FUNCTION_BLOCK RequestOrchestrationOpcUa (* Request Orchestration Function Block using OPC UA *)
  (* Standard: 61499-2; Description: Copyright (c) 2019 fortiss GmbH This program and the accompanying materials are made available under the terms of the Eclipse Public License 2.0 which is available at https://www.eclipse.org/legal/epl-2.0/ SPDX-License-Identifier: EPL-2.0 *)
  (* Version 1.0, 2019-09-17, Jose Cabral, fortiss GmbH *)
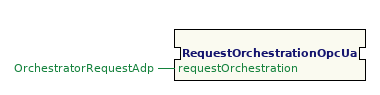
  SOCKETS
    requestOrchestration : OrchestratorRequestAdp; (* Request orchestration adapter *)
  END_SOCKETS
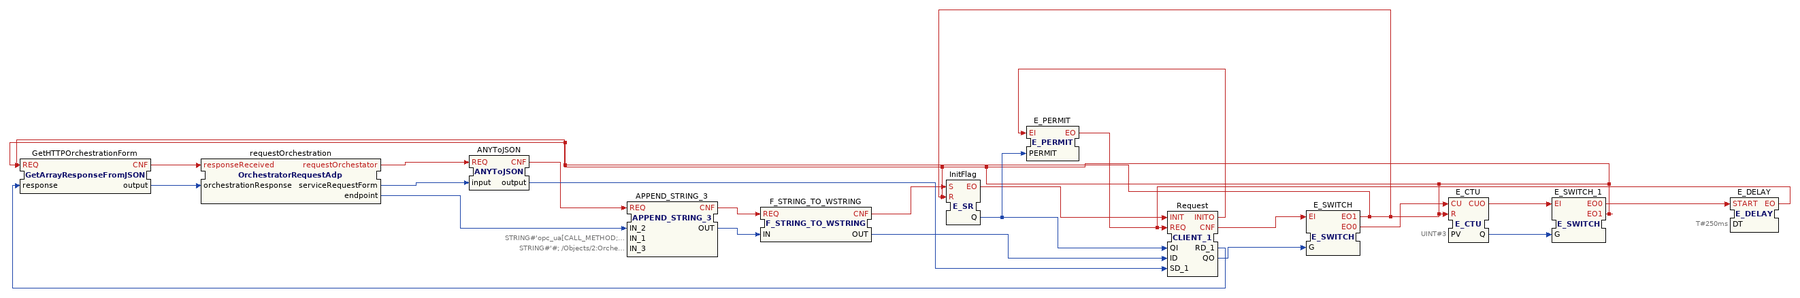
  FBS
    APPEND_STRING_3 : APPEND_STRING_3(IN_1 := STRING#'opc_ua[CALL_METHOD; ', IN_3 := STRING#'#; /Objects/2:Orchestrator/2:orchestration]');
    InitFlag : E_SR;
    E_PERMIT : E_PERMIT;
    F_STRING_TO_WSTRING : F_STRING_TO_WSTRING;
    ANYToJSON : ANYToJSON;
    GetHTTPOrchestrationForm : GetArrayResponseFromJSON;
    Request : CLIENT_1;
    E_SWITCH : E_SWITCH;
    E_SWITCH_1 : E_SWITCH;
    E_CTU : E_CTU(PV := UINT#3);
    E_DELAY : E_DELAY(DT := T#250ms);
  END_FBS
  EVENT_CONNECTIONS
    APPEND_STRING_3.CNF TO F_STRING_TO_WSTRING.REQ;
    F_STRING_TO_WSTRING.CNF TO InitFlag.S;
    ANYToJSON.CNF TO APPEND_STRING_3.REQ;
    requestOrchestration.requestOrchestator TO ANYToJSON.REQ;
    GetHTTPOrchestrationForm.CNF TO requestOrchestration.responseReceived;
    InitFlag.EO TO Request.INIT;
    E_PERMIT.EO TO Request.REQ;
    Request.INITO TO E_PERMIT.EI;
    E_SWITCH.EO1 TO GetHTTPOrchestrationForm.REQ;
    E_SWITCH.EO1 TO InitFlag.R;
    Request.CNF TO E_SWITCH.EI;
    E_SWITCH.EO0 TO E_CTU.CU;
    E_DELAY.EO TO Request.REQ;
    E_CTU.CUO TO E_SWITCH_1.EI;
    E_SWITCH_1.EO0 TO E_DELAY.START;
    E_SWITCH_1.EO1 TO InitFlag.R;
    E_SWITCH_1.EO1 TO GetHTTPOrchestrationForm.REQ;
    E_SWITCH.EO1 TO E_CTU.R;
    E_SWITCH_1.EO1 TO E_CTU.R;
  END_CONNECTIONS
  DATA_CONNECTIONS
    APPEND_STRING_3.OUT TO F_STRING_TO_WSTRING.IN;
    InitFlag.Q TO E_PERMIT.PERMIT;
    requestOrchestration.serviceRequestForm TO ANYToJSON.input;
    requestOrchestration.endpoint TO APPEND_STRING_3.IN_2;
    GetHTTPOrchestrationForm.output TO requestOrchestration.orchestrationResponse;
    InitFlag.Q TO Request.QI;
    F_STRING_TO_WSTRING.OUT TO Request.ID;
    ANYToJSON.output TO Request.SD_1;
    Request.RD_1 TO GetHTTPOrchestrationForm.response;
    Request.QO TO E_SWITCH.G;
    E_CTU.Q TO E_SWITCH_1.G;
  END_CONNECTIONS
END_FUNCTION_BLOCK
